Staubli VAL3: readData.pgx

program readData(sio& x_UdpSocket, num& x_nData[], bool& x_bNewData, bool& x_bError)
  local num l_nSioReadBytes
  local num l_nSioReadBytesBis
begin
  x_bNewData = false
  x_bError = false

  // Read from UDP socket
  l_nSioReadBytes = sioGet(x_UdpSocket, x_nData)

  if(l_nSioReadBytes == size(x_nData))
    // Successfully read a full message
    x_bNewData = true
    return
  elseIf (l_nSioReadBytes > 0)
    // Message of wrong size received, error
    logMsg("ros2_server::readData : message of wrong size received", 2)
    x_bError = true
    return
  endIf

  if (x_bNewData)
    // If we got something, try to read again to clear the buffer
    l_nSioReadBytesBis = sioGet(x_UdpSocket, x_nData)
  endIf

  if (l_nSioReadBytesBis > 0 and l_nSioReadBytesBis != size(x_nData))
    // Message of wrong size received, error
    logMsg("ros2_server::readData : message of wrong size received (2)", 2)
    x_bError = true
    return
  endIf

  // Check for errors
  if(l_nSioReadBytes == -1 or l_nSioReadBytesBis == -1)
    // Communication error of some kind
    x_bError = true
    logMsg("ros2_server::readData : Communication error", 2)
  elseIf(l_nSioReadBytes == 0)
    // No data available in buffer
    x_bError = false
    // logMsg("ros2_server::readData : No data available", 2)
  else
    // Communication error of some kind
    x_bError = true
    logMsg("ros2_server::readData : unexpected packet size", 2)
  endIf
end
